// TIA Portal V19 export
TYPE "JB_WeldingSetUp"
   STRUCT
      MaterialWidth : LReal;
      MeasureSheetEdgeReference : LReal;   // Distance of sheet edge from reference
      WeldingDirection : Bool;   // 0=towards to op (BKW=Minus) 1=away from op (FWD=Plus)
      CorrStartWelding : LReal;   // Start welding correction absolute value
      CorrStopWelding : LReal;   // Stop welding correction absolute value
   END_STRUCT;
END_TYPE
